TYPE ST_HMI_EquipmentStatus :
STRUCT
	Status : PackMLStates;
	Error : BOOL;
	Naam : STRING(30);
END_STRUCT
END_TYPE

(* stored: Version 1.1.0.1
   DUT ST_HMI_EquipmentStatus: Id {e7dfa1f1-b937-429c-a47d-c45f99d1d9ad} *)
